INTERFACE ITcoTaskStatus

PROPERTY Busy : BOOL
GET
END_GET
END_PROPERTY

PROPERTY Done : BOOL
GET
END_GET
END_PROPERTY

PROPERTY Error : BOOL
GET
END_GET
END_PROPERTY

END_INTERFACE

(* stored: Version 1.1.0.1
   Itf ITcoTaskStatus: Id {6341a5e9-539f-07e2-2781-89effa0ed565}
   Property Busy: Id {0f27cd62-9c61-0157-0eeb-42c4f74b66be}
   Get Get: Id {ae011746-e617-02b7-243e-e8509384b84f}
   Property Done: Id {e7e4f0d2-681c-0127-20a0-25e98eef98f1}
   Get Get: Id {ad228e2d-55b7-001f-0fb1-ccc8383b9be3}
   Property Error: Id {e997df47-5359-0431-0d62-646922dde6fe}
   Get Get: Id {1c91e88f-586c-08a8-3390-342071b85c00} *)
